SUBAPPLICATION Uebung_012g (* Numeric Value Input PHYS und Speichern INI *)
  (* Standard: 61499-2; Description: Copyright (c) 2023 Meisterschulen am Ostbahnhof This program and the accompanying materials are made available under the terms of the Eclipse Public License 2.0 which is available at https://www.eclipse.org/legal/epl-2.0/ SPDX-License-Identifier: EPL-2.0 *)
  (* Version 1.0, 2023-10-23, Franz Höpfinger, Meisterschulen am Ostbahnhof, initial API and implementation and/or initial documentation *)
  PACKAGE Uebungen;
  IMPORT Uebungen::const::NVS::NVS_Keys::KEY_I1_STORE;
  IMPORT Uebungen::const::UT::DefaultPool_Numeric::InputNumber_I3_N;
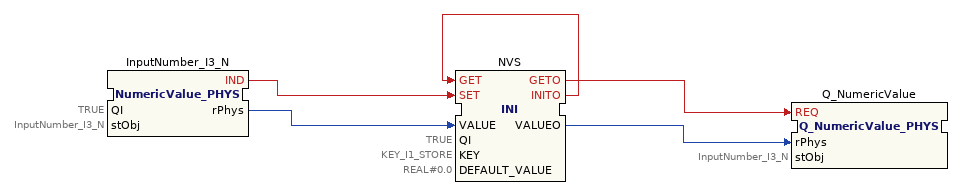
  FBS
    InputNumber_I3_N : isobus::UT::io::NumericValue::NumericValue_PHYS(QI := TRUE, stObj := InputNumber_I3_N);
    NVS : eclipse4diac::storage::INI(QI := TRUE, KEY := KEY_I1_STORE, DEFAULT_VALUE := REAL#0.0);
    Q_NumericValue : isobus::UT::Q::Q_NumericValue_PHYS(stObj := InputNumber_I3_N);
  END_FBS
  EVENT_CONNECTIONS
    NVS.GETO TO Q_NumericValue.REQ;
    NVS.INITO TO NVS.GET;
    InputNumber_I3_N.IND TO NVS.SET;
  END_CONNECTIONS
  DATA_CONNECTIONS
    NVS.VALUEO TO Q_NumericValue.rPhys;
    InputNumber_I3_N.rPhys TO NVS.VALUE;
  END_CONNECTIONS
END_SUBAPPLICATION
